FUNCTION "ASCF_CL_105_IF6" : Word
{ S7_Optimized_Access := 'TRUE' }
VERSION : 0.1
   VAR_OUTPUT
      Out : "ASCF_UnionType";
   END_VAR

   VAR_IN_OUT
      Arguments : Array[0..3] of "ASCF_UnionType";
      Memory : "ASCF_CL_ArgumentType";
   END_VAR

   VAR_TEMP
      Condition : Bool;
      Command : DWord;
      PrevResult : DWord;
      tempQCs : Array[0..3] of Byte;
      constDefaultUnionType : "ASCF_UnionType";
      constUnionTypes : "ASCF_EnumUnionTypes";
      constQualityCodes : "ASCF_QualityCodes";
      constSourceTypes : "ASCF_CL_EnumSourceTypes";
      constErrors : "ASCF_CL_EnumErrors";
   END_VAR


BEGIN


	REGION INITIALIZE VARIABLES

	    #Out := #constDefaultUnionType;

	END_REGION INITIALIZE VARIABLES

	REGION CHECK ARG0

	    IF #Memory.Source = #constSourceTypes.Constant THEN
	        #ASCF_CL_105_IF6 := #constErrors.InvalidSourceSelected;
	    END_IF;

	END_REGION CHECK ARG0

	REGION PROCESS ARGUMENTS


	    IF #Arguments[0].Typeselector <> #constUnionTypes.VBool THEN
	        #ASCF_CL_105_IF6 := #constErrors.InvalidType;
	        RETURN;
	    END_IF;

	    IF #Arguments[1].Typeselector <> #constUnionTypes.None THEN
	        #ASCF_CL_105_IF6 := #constErrors.InvalidType;
	        RETURN;
	    END_IF;

	    IF #Arguments[2].Typeselector <> #constUnionTypes.VDWord THEN
	        #ASCF_CL_105_IF6 := #constErrors.InvalidType;
	        RETURN;
	    END_IF;

	    IF #Arguments[3].Typeselector <> #constUnionTypes.VDWord THEN
	        #ASCF_CL_105_IF6 := #constErrors.InvalidType;
	        RETURN;
	    END_IF;

	    #Condition := #Arguments[0].VBool;
	    #Command := #Arguments[2].VDWord;
	    #PrevResult := #Arguments[3].VDWord;
	    #tempQCs[0] := #Arguments[0].VQC;
	    #tempQCs[1] := #constQualityCodes."No Status";
	    #tempQCs[2] := #Arguments[2].VQC;
	    #tempQCs[3] := #Arguments[3].VQC;

	END_REGION PROCESS ARGUMENTS

	REGION OUTPUT

	    #Out.VQC := "ASCF_CalcWQC"(QC1 := "ASCF_CalcWQC"(QC1 := #tempQCs[0], QC2 := #tempQCs[1]), QC2 := "ASCF_CalcWQC"(QC1 := #tempQCs[2], QC2 := #tempQCs[3]));
	    #Out.Typeselector := #constUnionTypes.VDWord;

	    IF NOT #Condition AND #Memory.Const.VBool THEN
	        #Out.VDWord := #Command;
	    ELSE
	        #Out.VDWord := #PrevResult;
	    END_IF;

	    #Memory.Const.VBool := #Condition;

	    #ASCF_CL_105_IF6 := #constErrors.None;

	END_REGION EXECUTE AND OUTPUT
END_FUNCTION